(* CODESYS project TSR Libary.library
   Company: Eaton Automation
   Title: TSR Libary
   Description: Das ist eine Libary die die Wichtigsten Funktionen für den Touch-Simulations Roboter berteitstellt.
   Author: Samuel A. Marti
   Version: 1.3

Project tree, tasks and I/O mapping:
  libraries: Standard, 3.5.2.0 (System); CAA SerialCom, 3.5.3.0 (CAA Technical Workgroup)
  POUs/
    TSR Com/
      function block TSR_Com [ST]: A00_Start, A01_Get_Settings, A02_Open_Com, A03_Open_Wait, A04_Send_Com, A05_Send_Wait, A06_Receive_Com, A07_Receive_Wait, A08_String_Auswertung, A09_End, B0100_Error, A10_Start, A13_End, B1100_Error, A12_Close_Wait, A11_Close_Com, A0_Port_Senden, A1_Port_Schliessen
    FB Connect with TSR/
      function block Connect_with_TSR [ST]: B100_Error, A00_Start, A01_Progress, A02_Progress_Wait, A03_Auswerten, A04_End, A10_Start, A11_Progress, A12_Progress_Wait, A13_Auswerten, A14_End, A0_Connect_with_TSR, A1_Disconnect_with_TSR
    FN Set TSR startpoint/
      function FN_Set_TSR_startpoint [ST]
    FB Move TSR xy/
      function block FB_Move_TSR_xy [ST]: A0_Start, A1_Progress, A2_Progress_Wait, A3_Auswerten, A4_Wait_for_TSR, A5_Wait_for_TSR_Wait, A6_Wait_for_TSR_Auswerten, A7_End, B100_Error
    FB Go to TSR xy/
      function block FB_Go_to_TSR_xy [ST]: A0_Start, A1_Progress, A2_Progress_Wait, A3_Auswerten, A4_Wait_for_TSR, A5_Wait_for_TSR_Wait, A6_Wait_for_TSR_Auswerten, A7_End, B100_Error
    FB Get TSR position/
      function block FB_Get_TSR_position [ST]: A0_Start, A1_Progress, A2_Progress_Wait, A3_Auswerten, A4_End, B100_Error
    FB TSR Pen up down/
      function block TSR_Pen_up_down [ST]: A0_Start, A1_Progress, A2_Progress_Wait, A3_Auswerten, A4_End, B100_Error
    FB Click/
      function block FB_Click [ST]: A0_Start, A1_Progress, A2_Progress_Wait, A3_PenDown, A4_PenDown_Wait, A5_PenUp, A6_PenUp_Wait, A7_End, B100_Error
    FB Double Click/
      function block FB_Double_Click [ST]: A0_Start, A1_Progress, A2_Progress_Wait, A3_PenDown, A4_PenDown_Wait, A5_PenUp, A6_PenUp_Wait, A7_End, B100_Error
  global variables GLOBAL
*)

// GLOBAL
VAR_GLOBAL
iStartPosx				:INT;			//Die Globale Variable des Neuen nulpunkts für die anderen FB's
iStartPosy				:INT;			//""
GTr_Faktor				:REAL := 8.8;	//Der umrechnungs Faktor: Momentan ist er auf mm abgestummen.
FB_TSRCom: 				TSR_Com;		//Die Com Communication
END_VAR

// POUs/TSR Com/TSR_Com
FUNCTION_BLOCK TSR_Com
VAR_INPUT									//FB Eingänge	
	xExecute				:BOOL;				//Startbedingung für den FB.
	iCom					:INT;				//Die Nummer des Com Ports.
	stSendData				:STRING;			//Der String der Gesendet werden soll.
	xPort					:BOOL;				//Wenn = 0 Wird der Port geschlossen, Wenn = 1 Wird der Port geöffnet.
END_VAR

VAR_OUTPUT									//FB Ausgänge
	xBusy					:BOOL;				//Das Busy bit.
	xDone					:BOOL;				//Ist 1 wenn FB fertig ist.
	stReceivedData			:STRING;			//Der Empfangene Daten String.
	wState					:WORD;				//Der ENUM Wert für die ENUM Tabelle.
	xError					:BOOL;				//Ist 1 wenn es einen Error gab.
END_VAR

VAR											//Interne Var
	LTi_Zustand				:INT;				//Der Zustand.
	LTi_PosString			:INT;				//Die Position vom Carisch retain lengfield.
	LTocpa_ComParameter1	:ARRAY[1..20] OF COM.PARAMETER; //Initalisierung der Com Parameter.
	
	LTx_ComOpen				:BOOL;				//Gibt an ob ein Com Port schon offen ist.
	LTudi_Handle			:UDINT;				//Der Interne COM Handle.
	LTst_ReceivedData		:STRING;			//Received Data zwischenspeicher.

	LTfb_ComOpen			:Com.Open;			//FB Open.
	LTfb_WriteCom			:Com.Write;			//FB Write.
	LTfb_ReadCom			:Com.Read;			//FB Read.
	LTfb_Close				:Com.Close;			//FB Für den Com port zu schliessen.
	LTfb_Timer				:TON;				//Timer Init.
	
	LTudi_ComPort			:UDINT;				//Welcher Com Port ist gemeint.

END_VAR

VAR CONSTANT								//Konstanten, Einstellungen
	LCudi_StopBit			:UDINT := 0;		//Die Stopbits: 0 = 1stb, 1 = 1.5stb, 2 = 2stb.
	LCudi_Parity			:UDINT := 2;		//Parity: 0 = gerade, 1 = ungerade, 2 = keine.
	LCudi_Baudrate			:UDINT := 9600; 	//Möglich sind 2,5 m 115200 Bit/s, 5 m 57600 Bit/s, 10 m 38400 Bit/s, 15 m 19200 Bit/s, 30 m 9600 Bit/s
	LCudi_TimeOut			:UDINT := 0;		//Keine ahnung was das bewirkt.
	LCudi_BufferSize		:UDINT := 2048;		//Die Buffer grösse.
	LCudi_ByteSize			:UDINT := 8;		//Die Grösse vom daten Byte. kann nur von 4 bis 8 sein
	LCudi_Binary			:UDINT := 0;		//Binärmodus, keine EOF-Überprüfung/ keine ahnung wad das ist.
	LCudi_OutxCTSFlow		:UDINT := 0;		//CTS Handshake auf Ausgang/ keine ahnung wad das ist.
	LCudi_OutxDSRFlow		:UDINT := 0; 		//DSR Handshake auf Ausgang/ keine ahnung wad das ist.
	LCudi_DTRControl		:UDINT := 0;		//DTR Control. DTR Flusssteuerung/ keine ahnung wad das ist.
	LCudi_DSRSensitiv		:UDINT := 0; 		//DSR Empfindlichkeit/ keine ahnung wad das ist.
	LCudi_RTSControl		:UDINT := 0;		//Rts Flussteuerung/ keine ahnung wad das ist.
	LCudi_TXContinueOnXoff	:UDINT := 0;		//XOFF fortfahren Tx / keine ahnung wad das ist.
	LCudi_OUTX				:UDINT := 0;		//XON/XOFF Ausgabeflusssteuerung / keine ahnung wad das ist.
	LCudi_INX				:UDINT := 0;		//XON/XOFF Eingabeflusssteuerung / keine ahnung wad das ist.
	LCudi_XOnChar			:UDINT := 0;		//Tx AND Rx XON Zeichen / keine ahnung wad das ist.
	LCudi_XOffChar			:UDINT := 0;		//Tx AND Rx XOFF Zeichen.
	LCudi_XOnLim			:UDINT := 0;		//Übertrage XON Schwellenwert
	LCudi_XOffLim			:UDINT := 0;		//Übertrage XOFF Schwellenwert
	
	LCt_WaitTimeout			:TIME := T#4S;			//der Timout Timer.
	LCt_WaitCom				:TIME := T#600MS;		//Wait auf Received Data.
END_VAR

IF xPort = 1 THEN
	A0_Port_Senden();
END_IF

IF xPort = 0 THEN
	A1_Port_Schliessen();
END_IF

LTfb_Close();
LTfb_ComOpen();

ACTION A00_Start:
IF xExecute THEN			//Prüfe Startbedinung.
	xBusy := 1;				//Setze Busy.
	IF LTx_ComOpen THEN 	//Ist der Com Port offen ?
		LTi_Zustand := 4;	//Gehe direkt zum Schritt wo der String geschrieben wird.
	ELSE
		LTi_Zustand := 1;	//Gehe direkt zum Schritt wo der Com Port geöffnet wird.
	END_IF
END_IF
END_ACTION

ACTION A01_Get_Settings:
LTudi_ComPort := INT_TO_UDINT(iCom);

//Port
LTocpa_ComParameter1[1].udiParameterId := COM.CAA_Parameter_Constants.udiPort;		//ID von Com Port
LTocpa_ComParameter1[1].udiValue := LTudi_ComPort;									//Der COM Port1

//Stopbit
LTocpa_ComParameter1[2].udiParameterId := COM.CAA_Parameter_Constants.udiStopBits;	//ID von StopBit
LTocpa_ComParameter1[2].udiValue := LCudi_StopBit;									//Der COM Port. 0 = 1stb, 1 = 1.5stb, 2 = 2stb.

//Parität
LTocpa_ComParameter1[3].udiParameterId := COM.CAA_Parameter_Constants.udiParity;		//ID von Parity
LTocpa_ComParameter1[3].udiValue := LCudi_Parity;									//0 = gerade, 1 = ungerade, 2 = keine.

//Baudrate
LTocpa_ComParameter1[4].udiParameterId := COM.CAA_Parameter_Constants.udiBaudrate;	//ID von Baudrate
LTocpa_ComParameter1[4].udiValue := LCudi_Baudrate;									//Möglich sind 2,5 m 115200 Bit/s, 5 m 57600 Bit/s, 10 m 38400 Bit/s, 15 m 19200 Bit/s, 30 m 9600 Bit/s

//Timeout
LTocpa_ComParameter1[5].udiParameterId := COM.CAA_Parameter_Constants.udiTimeout;	//ID von Timeout
LTocpa_ComParameter1[5].udiValue := LCudi_TimeOut;									//Keine ahnung wad das ist.
(*
//BufferSize																		
LTocpa_ComParameter1[6].udiParameterId := COM.CAA_Parameter_Constants.udiBufferSize;	//ID von Buffersize
LTocpa_ComParameter1[6].udiValue := GLRudi_BufferSize;								//Die Grösse die der Buffer haben soll
*)
//ByteSize																	
LTocpa_ComParameter1[7].udiParameterId := COM.CAA_Parameter_Constants.udiByteSize;	//ID von ByteSize
LTocpa_ComParameter1[7].udiValue := LCudi_ByteSize;									//Die Grösse vom daten Byte. kann nur von 4 bis 8 sein

//Binary
LTocpa_ComParameter1[8].udiParameterId := COM.CAA_Parameter_Constants.udiBinary;	//ID von Binary
LTocpa_ComParameter1[8].udiValue := LCudi_Binary;									//Binärmodus, keine EOF-Überprüfung/ keine ahnung wad das ist.
(*
//OutxCtsFlow
LTocpa_ComParameter1[9].udiParameterId := COM.CAA_Parameter_Constants.udiOutxCtsFlow;	//ID von OutxCtsFlow
LTocpa_ComParameter1[9].udiValue := LCudi_OutxCTSFlow;									//CTS Handshake auf Ausgang/ keine ahnung wad das ist.

//OutxDSRFlow
LTocpa_ComParameter1[10].udiParameterId := COM.CAA_Parameter_Constants.udiOutxDsrFlow;	//ID von OutxDSRFlow
LTocpa_ComParameter1[10].udiValue := LCudi_OutxDSRFlow;									//DSR Handshake auf Ausgang/ keine ahnung wad das ist.

//DTRControl
LTocpa_ComParameter1[11].udiParameterId := COM.CAA_Parameter_Constants.udiDtrControl;	//ID von DtrControl
LTocpa_ComParameter1[11].udiValue := LCudi_OutxDSRFlow;									//DSR Handshake auf Ausgang/ keine ahnung wad das ist.

//DSR Sensitiv
LTocpa_ComParameter1[12].udiParameterId := COM.CAA_Parameter_Constants.udiDsrSensitivity;//ID von DSR Sensitiv
LTocpa_ComParameter1[12].udiValue := LCudi_DSRSensitiv;									//DSR Empfindlichkeit/ keine ahnung wad das ist.

//RTS Control
LTocpa_ComParameter1[13].udiParameterId := COM.CAA_Parameter_Constants.udiRtsControl;	//ID von RTS Control
LTocpa_ComParameter1[13].udiValue := LCudi_RTSControl;									//Rts Flusssteuerung/ keine ahnung wad das ist.

//TXContinueOnXoff	
LTocpa_ComParameter1[14].udiParameterId := COM.CAA_Parameter_Constants.udiTXContinueOnXoff;	//ID von  XOFF fortfahren Tx	
LTocpa_ComParameter1[14].udiValue := LCudi_TXContinueOnXoff;									//XOFF fortfahren Tx / keine ahnung wad das ist.

//OUT X
LTocpa_ComParameter1[15].udiParameterId := COM.CAA_Parameter_Constants.udiOutX;	//ID von OUT X	
LTocpa_ComParameter1[15].udiValue := LCudi_OUTX;									//XON/XOFF Ausgabeflusssteuerung/ keine ahnung wad das ist.

//IN X
LTocpa_ComParameter1[16].udiParameterId := COM.CAA_Parameter_Constants.udiInX;	//ID von IN X	
LTocpa_ComParameter1[16].udiValue := LCudi_INX;									//Eingabeflusssteuerung/ keine ahnung wad das ist.

//XOnChar
LTocpa_ComParameter1[17].udiParameterId := COM.CAA_Parameter_Constants.udiXonChar;	//ID von x on char	
LTocpa_ComParameter1[17].udiValue := LCudi_XOnChar;									//Tx AND Rx XON Zeichen/ keine ahnung wad das ist.

//XOffChar
LTocpa_ComParameter1[18].udiParameterId := COM.CAA_Parameter_Constants.udiXoffChar;	//ID von x off char
LTocpa_ComParameter1[18].udiValue := LCudi_XOffChar;									//Tx AND Rx XOFF Zeichen/ keine ahnung wad das ist.

//XonLim
LTocpa_ComParameter1[19].udiParameterId := COM.CAA_Parameter_Constants.udiXonLim;	//ID von X on Lim
LTocpa_ComParameter1[19].udiValue := LCudi_XOnLim;									//Übertrage XON Schwellenwert/ keine ahnung wad das ist.

//XoffLim
LTocpa_ComParameter1[20].udiParameterId := COM.CAA_Parameter_Constants.udiXonLim;	//ID von X off Lim
LTocpa_ComParameter1[20].udiValue := LCudi_XOnLim;									//Übertrage XOFF Schwellenwert/ keine ahnung wad das ist.
*)
LTi_Zustand := 2;
END_ACTION

ACTION A02_Open_Com:
//Com Port öffnen
LTfb_ComOpen.usiListLength := INT_TO_USINT(SIZEOF(LTocpa_ComParameter1));	//Die länge der Parameter Liste
LTfb_ComOpen.pParameterList := ADR(LTocpa_ComParameter1);		//Die Adresse der Parameter Liste
LTfb_ComOpen.xExecute := 1;									//Start Flag setzten.
LTi_Zustand := 3;
LTfb_Timer(IN := 1, PT:= LCt_WaitTimeout);								//Rufe Timer auf
END_ACTION

ACTION A03_Open_Wait:
IF LTfb_ComOpen.xDone THEN											//Wenn der Port offen
	LTfb_Timer.IN := 0;					//Timer Zurücksetzten.
	LTi_Zustand := 4;					//Gehe in den Sende Schritt
	LTudi_Handle := LTfb_ComOpen.hCom;	//Speichere den Handle
	LTx_ComOpen	:= 1;					//Der Offene Com Port setzten.
ELSE
	IF LTfb_ComOpen.xError THEN				//Wenn es einen Error bei Com Port öffnen gab.
		LTfb_Timer.IN := 0;					//Timer Zurücksetzten.
		LTi_Zustand := 100;					//In den Error Zustand gehen.
		wState := 1;						//Den ENUM Wert Error angeben.
	ELSE
		IF LTfb_Timer.Q THEN						//Wenn der Timer Abgelaufen ist.
			LTi_Zustand := 100;					//In den Error Zustand gehen.
			wState := 4;						//Den ENUM Wert Error angeben.
			LTfb_Timer.IN := 0;
		END_IF
	END_IF
END_IF

LTfb_Timer();								//Rufe Timer auf
LTfb_ComOpen();							//Rufe den FB auf.
END_ACTION

ACTION A04_Send_Com:
LTfb_WriteCom(
	hCom			:= LTudi_Handle, 						//Ubergebe Handle.
	pBuffer 		:= ADR(stSendData),
	szSize 			:= INT_TO_UDINT(SIZEOF(stSendData)),
	xExecute		:= 1									//Starte Sende Vorgang.
);

LTi_Zustand := 5;
LTfb_Timer(IN := 1, PT:= LCt_WaitTimeout);				//Rufe Timer auf
END_ACTION

ACTION A05_Send_Wait:
IF LTfb_WriteCom.xDone THEN				//Wenn der String gesendet wurde.
	LTfb_Timer.IN := 0;					//Timer Zurücksetzten.
	LTi_Zustand := 6;					//Gehe in den Sende Schritt
ELSE
	IF LTfb_WriteCom.xError THEN				//Wenn es einen Error bei String senden gab.
		LTfb_Timer.IN := 0;					//Timer Zurücksetzten.
		LTi_Zustand := 100;					//In den Error Zustand gehen.
		wState := 2;						//Den ENUM Wert Error angeben.
	ELSE
		IF LTfb_Timer.Q THEN						//Wenn der Timer Abgelaufen ist.
			LTi_Zustand := 100;					//In den Error Zustand gehen.
			wState := 5;						//Den ENUM Wert Error angeben.
			LTfb_Timer.IN := 0;
		END_IF
	END_IF
END_IF

LTfb_Timer();								//Rufe Timer auf
LTfb_WriteCom();							//Rufe den FB auf.
END_ACTION

ACTION A06_Receive_Com:
LTfb_Timer(IN := 1, PT:= LCt_WaitCom);			//Rufe Timer auf
IF LTfb_TIMER.Q THEN							//Wenn der Timer fertig ist
	LTfb_Timer.IN := 0;						//Timer zurücksetzten
	LTfb_Timer();								//FB Timer zurückstzen.
	
	LTfb_ReadCom								//Rufe ReadCom auf.
	(
		xExecute	:= 1,					//Starte Lese STRING
		hCom		:= LTudi_Handle,		//übergib den Handle.
		pBuffer := ADR(LTst_ReceivedData),
		szBuffer := SIZEOF(LTst_ReceivedData),
	);
LTi_Zustand := 7;

END_IF
END_ACTION

ACTION A07_Receive_Wait:
IF LTfb_ReadCom.xDone THEN				//Wenn der String gesendet wurde.
	LTfb_Timer.IN := 0;					//Timer Zurücksetzten.
	LTi_Zustand := 8;					//Gehe in den Sende Schritt
ELSE
	IF LTfb_ReadCom.xError THEN				//Wenn es einen Error bei String senden gab.
		LTfb_Timer.IN := 0;					//Timer Zurücksetzten.
		LTi_Zustand := 100;					//In den Error Zustand gehen.
		wState := 3;						//Den ENUM Wert Error angeben.
	ELSE
		IF LTfb_Timer.Q THEN						//Wenn der Timer Abgelaufen ist.
			LTi_Zustand := 100;					//In den Error Zustand gehen.
			wState := 6;						//Den ENUM Wert Error angeben.
			LTfb_Timer.IN := 0;
		END_IF
	END_IF
LTfb_Timer(IN := 1, PT:= LCt_WaitTimeout);			//Schalte Timer ein.
END_IF

LTfb_Timer();								//Rufe Timer auf
LTfb_ReadCom();							//Rufe den FB auf.
END_ACTION

ACTION A08_String_Auswertung:
LTi_PosString := FIND(STR2:='$R$N' , STR1:=LTst_ReceivedData);		//Das caretsch Retain lengfield 
LTst_ReceivedData[LTi_PosString - 1] := 0;							//DAs caretain legas löschen mit allem was dahinter ist.
stReceivedData := LTst_ReceivedData;								//Ausgeben
LTi_Zustand := 9;													//Zum Zustand 9 gehen.
END_ACTION

ACTION A09_End:
xBusy := 0;							//Alles zurücksetzten
xDone := 1;
IF xExecute = 0 THEN				//Warten bis der User Zurückgesetzt hat.
	xDone := 0;
	LTi_Zustand := 0;
	stReceivedData := '';
	LTfb_WriteCom.xExecute := 0;
	LTfb_ReadCom.xExecute := 0;
	LTst_ReceivedData := '';
	LTfb_ComOpen.xExecute := 0;
	LTfb_WriteCom();
	LTfb_ReadCom();
	LTfb_ComOpen();
END_IF
END_ACTION

ACTION B0100_Error:
xBusy := 0;							//Alles zurücksetzten
xError := 1;
IF xExecute = 0 THEN				//Wartem bis der User das xExecute zurückgesetzt hat.
	xError := 0;
	LTi_Zustand := 0;
	wState := 0;
	stReceivedData := '';
	LTst_ReceivedData := '';
	LTfb_WriteCom.xExecute := 0;
	LTfb_ReadCom.xExecute := 0;
	LTfb_ComOpen.xExecute := 0;
	LTfb_WriteCom();
	LTfb_ReadCom();
	LTfb_ComOpen();
END_IF
END_ACTION

ACTION A10_Start:
IF xExecute THEN			//Prüfe Startbedinung.
	xBusy := 1;				//Setze Busy.
	IF LTx_ComOpen THEN 	//Ist der Com Port offen ?
		LTi_Zustand := 1;	//Gehe direkt zum Schritt wo der String geschrieben wird.
	ELSE
		LTi_Zustand := 100; //Gehe in den Error Mod
		wState := 13;		//Bedeutung: Der com port ist nicht offen daher kann nichts geschlossen werden. 		
	END_IF
END_IF
END_ACTION

ACTION A13_End:
xBusy := 0;							//Alles zurücksetzten
xDone := 1;
IF xExecute = 0 THEN				//Warten bis der User Zurückgesetzt hat.
	xDone := 0;
	LTi_Zustand := 0;
	stReceivedData := '';
	LTst_ReceivedData := '';
	LTfb_Close.xExecute := 0;
	LTfb_Close();
END_IF
END_ACTION

ACTION B1100_Error:
xBusy := 0;							//Alles zurücksetzten
xError := 1;
IF xExecute = 0 THEN				//Wartem bis der User das xExecute zurückgesetzt hat.
	xError := 0;
	LTi_Zustand := 0;
	wState := 0;
	stReceivedData := '';
	LTst_ReceivedData := '';
	LTfb_Close.xExecute := 0;
	LTfb_Close();
END_IF
END_ACTION

ACTION A12_Close_Wait:
IF LTfb_Close.xDone THEN											//Wenn der Port offen
	LTfb_Timer.IN := 0;					//Timer Zurücksetzten.
	LTi_Zustand := 3;					//Gehe in den Finish schritt.
	LTx_ComOpen := 0;					//Denn Das Com Port flag zurücksetzten.
ELSE
	IF LTfb_Close.xError THEN				//Wenn es einen Error bei Com Port öffnen gab.
		LTfb_Timer.IN := 0;					//Timer Zurücksetzten.
		LTi_Zustand := 100;					//In den Error Zustand gehen.
		wState := 23;						//Den ENUM Wert Error angeben.
	ELSE
		IF LTfb_Timer.Q THEN						//Wenn der Timer Abgelaufen ist.
			LTi_Zustand := 100;					//In den Error Zustand gehen.
			wState := 24;						//Den ENUM Wert Error angeben.
			LTfb_Timer.IN := 0;
		END_IF
	END_IF
END_IF

LTfb_Timer();								//Rufe Timer auf
LTfb_ComOpen();							//Rufe den FB auf.
END_ACTION

ACTION A11_Close_Com:
LTfb_Close
(
	xExecute := 1 , 			//Setzt den Zustand vom Execute auf 1.
	hCom := LTudi_Handle, 		//übergebe den Handle des geöffneten Com Ports.
);
LTi_Zustand := 2;
END_ACTION

ACTION A0_Port_Senden:
CASE LTi_Zustand OF
	0:
		A00_Start();					//Prüfe die Startbedingungen und Prüfe auf einen offenen Com Port
	1:
		A01_Get_Settings();			//Holt die Einstellungen für zu öffnenden Com Port.
	2:
		A02_Open_Com();				//Öffnet den Com Port.
	3:
		A03_Open_Wait();				//Wartet bis der Com Port offen ist.
	4:
		A04_Send_Com();				//Den String Senden.
	5:
		A05_Send_Wait();				//Warte bis der String gesendet wurde.
	6:
		A06_Receive_Com();			//Empfange den String.
	7:
		A07_Receive_Wait();			//Warte auf FB String lesen.
	8:
		A08_String_Auswertung();		//Werte den FB String aus.
	9:
		A09_End();					//Beende den FB vorgang und warte auf das zurücksetzten.
	100:
		B0100_Error();				//Nur wenn ein Error gab.
END_CASE

LTfb_ComOpen();
END_ACTION

ACTION A1_Port_Schliessen:
CASE LTi_Zustand OF
	0:
		A10_Start();					//Prüfe die Startbedingungen und Prüfe auf einen offenen Com Port.
	1:
		A11_Close_Com();				//schliesst den Com Port.
	2:
		A12_Close_Wait();				//Warten bis der Com Port geschlossen.
	3:
		A13_End();						//Beendet den schliess vorgang.
	100:
		B1100_Error();					//Der Error Modus.
END_CASE

LTfb_Close();
END_ACTION

END_FUNCTION_BLOCK

// POUs/FB Connect with TSR/Connect_with_TSR
FUNCTION_BLOCK Connect_with_TSR
VAR_INPUT								//FB Eingänge
	xExecute				:BOOL;			//Startbedingung für den FB.
	iCom					:INT;			//Die Nummer des Com Ports.
	xPort					:BOOL;			//Bei 0 = den Port schliessen, bei 1 = Prot öffnen.
END_VAR

VAR_OUTPUT								//FB Ausgänge	
	xBusy					:BOOL;			//Das Busy bit.
	xDone					:BOOL;			//Ist 1 wenn FB fertig ist.
	wState					:WORD;			//Der ENUM Wert für die ENUM Tabelle.
	xError					:BOOL;			//Ist 1 wenn es einen Error gab.
END_VAR

VAR										//Interne Vars
	LTi_Zustand				:INT;			//Der Zustand.
	GLfb_Timer				:TON;			//Timer Init
END_VAR

VAR CONSTANT							//Konstanten, Einstellungen
	LCt_WaitTimeout			:TIME := T#4S;	//der Timout Timer. Nach welcher Zeit soll es einen Timeout geben.
END_VAR

//Entscheiden ob der COM Port geöffnent werden soll oder geschlossen werden soll
IF xPort = 0 THEN
	A1_Disconnect_with_TSR();	//Verbindung Abbrechen
END_IF

IF xPort = 1 THEN
	A0_Connect_with_TSR();		//Verbindung herstellen
END_IF
FB_TSRCom();

ACTION B100_Error:
xBusy := 0;							//Alles zurücksetzten
xError := 1;
IF xExecute = 0 THEN				//Wartem bis der User das xExecute zurückgesetzt hat.
	xError := 0;
	LTi_Zustand := 0;
	wState := 0;
	FB_TSRCom.xEXecute := 0;
END_IF
END_ACTION

ACTION A00_Start:
IF xExecute THEN			//Prüfe Startbedinung.
	xBusy := 1;				//Setze Busy.
	LTi_Zustand := 1;	//Gehe direkt zum Schritt wo der Com Port geöffnet wird.
END_IF
END_ACTION

ACTION A01_Progress:
FB_TSRCom(						//TSR Com Aufrufen und Daten übergeben.
	xEXecute	:=	1 , 
	xPort		:=	xPort,
	iCom		:= 	iCom, 
	stSendData	:= 	'?',  );
LTi_Zustand := 2;				//In den nächsten Zustand Wechseln.
END_ACTION

ACTION A02_Progress_Wait:
IF FB_TSRCom.xDone THEN											//Wenn der Port offen
	GLfb_Timer.IN := 0;					//Timer Zurücksetzten.
	LTi_Zustand := 3;					//Gehe in den Sende Schritt
ELSE
	IF FB_TSRCom.xError THEN				//Wenn es einen Error bei Com Port öffnen gab.
		GLfb_Timer.IN := 0;					//Timer Zurücksetzten.
		LTi_Zustand := 100;					//In den Error Zustand gehen.
		wState := FB_TSRCom.wState;			//Den ENUM Wert Error angeben.
	ELSE
		IF GLfb_Timer.Q THEN						//Wenn der Timer Abgelaufen ist.
			LTi_Zustand := 100;					//In den Error Zustand gehen.
			wState := 16;						//Timeout beim Connect
			GLfb_Timer.IN := 0;
		END_IF
	END_IF
GLfb_Timer(IN := 1, PT:= LCt_WaitTimeout);
END_IF

GLfb_Timer();								//Rufe Timer auf
END_ACTION

ACTION A03_Auswerten:
IF FB_TSRCom.stReceivedData = '!' THEN		//Wenn der TSR reagiert.
	LTi_Zustand := 4;						//Gehe zum letzten Zustand.
ELSE											
	LTi_Zustand := 100;	
	wState := 8;								
END_IF
END_ACTION

ACTION A04_End:
xBusy := 0;							//Alles zurücksetzten
xDone := 1;
IF xExecute = 0 THEN				//Warten bis der User Zurückgesetzt hat.
	xDone := 0;
	LTi_Zustand := 0;
	FB_TSRCom.xEXecute := 0;
END_IF
END_ACTION

ACTION A10_Start:
IF xExecute THEN			//Prüfe Startbedinung.
	xBusy := 1;				//Setze Busy.
	LTi_Zustand := 1;	//Gehe direkt zum Schritt wo der Com Port geöffnet wird.
END_IF
END_ACTION

ACTION A11_Progress:
FB_TSRCom(						//TSR Com Aufrufen und Daten übergeben.
	xEXecute	:=	1 , 
	iCom		:= 	iCom, 
	xPort		:=	xPort, );
LTi_Zustand := 2;				//In den nächsten Zustand Wechseln.
END_ACTION

ACTION A12_Progress_Wait:
IF FB_TSRCom.xDone THEN											//Wenn der Port offen
	GLfb_Timer.IN := 0;					//Timer Zurücksetzten.
	LTi_Zustand := 3;					//Gehe in den Sende Schritt
ELSE
	IF FB_TSRCom.xError THEN				//Wenn es einen Error bei Com Port öffnen gab.
		GLfb_Timer.IN := 0;					//Timer Zurücksetzten.
		LTi_Zustand := 100;					//In den Error Zustand gehen.
		wState := FB_TSRCom.wState;			//Den ENUM Wert Error angeben.
	ELSE
		IF GLfb_Timer.Q THEN					//Wenn der Timer Abgelaufen ist.
			LTi_Zustand := 100;					//In den Error Zustand gehen.
			wState := 16;						//Timeout_beim_Connect_weahrend_dem_TSR_COM
			GLfb_Timer.IN := 0;
		END_IF
	END_IF
GLfb_Timer(IN := 1, PT:= LCt_WaitTimeout);
END_IF

GLfb_Timer();								//Rufe Timer auf
END_ACTION

ACTION A13_Auswerten:
IF FB_TSRCom.stReceivedData = '' THEN		//Wenn der TSR reagiert.
	LTi_Zustand := 4;						//Gehe zum letzten Zustand.
ELSE											
	LTi_Zustand := 100;	
	wState := 8;								
END_IF
END_ACTION

ACTION A14_End:
xBusy := 0;							//Alles zurücksetzten
xDone := 1;
IF xExecute = 0 THEN				//Warten bis der User Zurückgesetzt hat.
	xDone := 0;
	LTi_Zustand := 0;
	FB_TSRCom.xEXecute := 0;
END_IF
END_ACTION

ACTION A0_Connect_with_TSR:
CASE LTi_Zustand OF
	0:
		A00_Start();					//Prüfe die Startbedingungen 
	1:
		A01_Progress();				//Starte den Prozess.
	2:
		A02_Progress_Wait();			//Warte auf den FB TSR Com
	3:
		A03_Auswerten();				//Werte das Egebniss aus.
	4:
		A04_End();					//Warte auf Execute
	100:
		B100_Error();				//Nur wenn ein Error gab.
END_CASE
END_ACTION

ACTION A1_Disconnect_with_TSR:
CASE LTi_Zustand OF
	0:
		A10_Start();					//Prüfe die Startbedingungen 
	1:
		A11_Progress();				//Starte den Prozess.
	2:
		A12_Progress_Wait();			//Warte auf den FB TSR Com
	3:
		A13_Auswerten();				//Werte das Egebniss aus.
	4:
		A14_End();					//Warte auf Execute
	100:
		B100_Error();				//Nur wenn ein Error gab.
END_CASE
END_ACTION

END_FUNCTION_BLOCK

// POUs/FN Set TSR startpoint/FN_Set_TSR_startpoint
FUNCTION FN_Set_TSR_startpoint : BOOL
VAR_INPUT							//FB EINGANGS VAR
	iStartpointx			:INT;		//Der Virtuelle x Nullpunkt.
	iStartpointy			:INT;		//Der Virtuelle y Nullpunkt.
END_VAR

iStartPosx := REAL_TO_INT(INT_TO_REAL(iStartpointx) * GTr_Faktor);		//Speicher eingang in Global Var
iStartPosy := REAL_TO_INT(INT_TO_REAL(iStartpointy) * GTr_Faktor);		//Speicher eingang in Global Var
FN_Set_TSR_startpoint := 1;												// Der Rückgabe wert der Funktion

END_FUNCTION

// POUs/FB Move TSR xy/FB_Move_TSR_xy
FUNCTION_BLOCK FB_Move_TSR_xy
VAR_INPUT									//Eingänge Var						
	xExecute				:BOOL;				//Startbedingung für den FB.
	iMovx					:INT;				//Die relative x bewegung des TSR in richtung x
	iMovy					:INT;				//Die relative y bewegung des TSR in richtung y
END_VAR

VAR_OUTPUT									//Ausgänge Var
	xBusy					:BOOL;				//Das Busy bit.
	xDone					:BOOL;				//Ist 1 wenn FB fertig ist.
	wState					:WORD;				//Der ENUM Wert für die ENUM Tabelle.
	xError					:BOOL;				//Ist 1 wenn es einen Error gab.
END_VAR

VAR											//Interne Var
	LTi_Zustand				:INT;				//Der Zustand.
	LTst_Zwischenspeicher	:STRING;			//Ein Zwischenspeicher für den Progress.
	LTi_Len					:INT;				//Gibt die String länge an für den Progress.
	LTi_x					:INT;				//Die x Schritte die der TSR machen soll.
	LTi_y					:INT;				//Die y Schritte die der TSR machen soll.
											//TIMER
	FN_Timer				:TON;				//Timer Init.
END_VAR

VAR CONSTANT								//Konstanten, Einstellungen
	LCt_WaitTimeout			:TIME := T#2S;		//der Timout Timer.
	LCt_WaitCom				:TIME := T#250MS;	//Wait auf Received Data.
END_VAR

CASE LTi_Zustand OF
	0:
		A0_Start();						//Prüfe Startbedingunen
	1:
		A1_Progress();					//Starte den Prozess. und sende den Befehl an das TSR.
	2:
		A2_Progress_Wait();				//Warte auf den FB Com.
	3:
		A3_Auswerten();					//Beende den FB und warte auf den User.
	4:
		A4_Wait_for_TSR();				//Init warten bis der TSR bei der Position angekommen ist
	5:
		A5_Wait_for_TSR_Wait();			//Warte auf FB Com.
	6:
		A6_Wait_for_TSR_Auswerten();	//Werte aus.
	7:
		A7_End();						//Das ende der Funktion.
	100:
		B100_Error();					//Die Error Aktion.
END_CASE

FB_TSRCom();							//Aufrufen.

ACTION A0_Start:
IF xExecute THEN			//Prüfe Startbedinung.
	xBusy := 1;				//Setze Busy.
	LTi_Zustand := 1;		//nächster Schritt
END_IF
END_ACTION

ACTION A1_Progress:
//Hier wird der Befehl für den TSR zusammengesetzt.
LTst_Zwischenspeicher := 'mov ';	//Speicher

//Die Fakto miteinbeziehen so das die mm umgerechnet werden, in Schritte.
LTi_x := REAL_TO_INT(INT_TO_REAL(iMovx) * GTr_Faktor);
//Schreibe Die X koordinate hinein.
LTst_Zwischenspeicher := INSERT(LTst_Zwischenspeicher,INT_TO_STRING(LTi_x),4); 

//Finde die länge des String heraus
LTi_Len := LEN(STR := LTst_Zwischenspeicher);

//Schreibe am Schluss ein :
LTst_Zwischenspeicher := INSERT(LTst_Zwischenspeicher,':',LTi_Len);

//Die Fakto miteinbeziehen so das die mm umgerechnet werden, in Schritte.
LTi_y := REAL_TO_INT(INT_TO_REAL(iMovy) * GTr_Faktor);
//Nun schreibe hinter dem : die y Koordiante.
LTst_Zwischenspeicher := INSERT(LTst_Zwischenspeicher,INT_TO_STRING(LTi_y),(LTi_Len + 1));

//TSR Com Aufrufen und Daten übergeben.
FB_TSRCom(						
	iCom		:= 1,
	xEXecute	:=	1 , 
	stSendData	:= 	LTst_Zwischenspeicher,  );

//Auf zum nächsten schritt.
LTi_Zustand := 2;
END_ACTION

ACTION A2_Progress_Wait:
IF FB_TSRCom.xDone THEN											//Wenn der Port offen
	FN_Timer.IN := 0;						//Timer Zurücksetzten.
	LTi_Zustand := 3;						//Gehe in den Sende Schritt
ELSE
	IF FB_TSRCom.xError THEN				//Wenn es einen Error bei Com Port öffnen gab.
		FN_Timer.IN := 0;					//Timer Zurücksetzten.
		LTi_Zustand := 100;					//In den Error Zustand gehen.
		wState := FB_TSRCom.wState;			//Den ENUM Wert Error angeben.
	ELSE
		IF FN_Timer.Q THEN					//Wenn der Timer Abgelaufen ist.
			LTi_Zustand := 100;				//In den Error Zustand gehen.
			wState := 21;					//Den ENUM Wert Error angeben.
			FN_Timer.IN := 0;
		END_IF
	END_IF
FN_Timer(IN := 1, PT:= LCt_WaitTimeout);	//Setzte den Timer.
END_IF
FN_Timer();									//Timer Aufrufen.
END_ACTION

ACTION A3_Auswerten:
IF FB_TSRCom.stReceivedData = 'moving' THEN //Wenn der TSR reagiert.
	LTi_Zustand := 4;						//Gehe zum letzten Zustand.
	FB_TSRCom.xEXecute := 0;				//Setzte Com Communication zurück.
ELSE
	IF FB_TSRCom.stReceivedData = 'out of range' THEN
		wState := 9;						//out of range state
		LTi_zustand := 100;
	ELSE
		LTi_Zustand := 100;
		wState := 8;							//Gehe zum letzten Zustand.
	END_IF
END_IF
END_ACTION

ACTION A4_Wait_for_TSR:
//TSR Com Aufrufen und Daten übergeben.
FB_TSRCom(						
	iCom		:= 1,
	xEXecute	:=	1 , 
	stSendData	:= 'state',  );				//frage den Status ab.

//Auf zum nächsten schritt.
LTi_Zustand := 5;
END_ACTION

ACTION A5_Wait_for_TSR_Wait:
IF FB_TSRCom.xDone THEN											//Wenn der Port offen
	FN_Timer.IN := 0;						//Timer Zurücksetzten.
	LTi_Zustand := 6;						//Gehe in den Sende Schritt
ELSE
	IF FB_TSRCom.xError THEN				//Wenn es einen Error bei Com Port öffnen gab.
		FN_Timer.IN := 0;					//Timer Zurücksetzten.
		LTi_Zustand := 100;					//In den Error Zustand gehen.
		wState := FB_TSRCom.wState;			//Den ENUM Wert Error angeben.
	ELSE
		IF FN_Timer.Q THEN					//Wenn der Timer Abgelaufen ist.
			LTi_Zustand := 100;				//In den Error Zustand gehen.
			wState := 21;					//Den ENUM Wert Error angeben.
			FN_Timer.IN := 0;
		END_IF
	END_IF
FN_Timer(IN := 1, PT:= LCt_WaitTimeout);	//Setzte den Timer.
END_IF
FN_Timer();									//Timer Aufrufen.
END_ACTION

ACTION A6_Wait_for_TSR_Auswerten:
IF FB_TSRCom.stReceivedData = 'ready' THEN 		//Wenn der TSR reagiert.
	LTi_Zustand := 7;							//Gehe zum letzten Zustand.
	FB_TSRCom.xEXecute := 0;					//Setzte Com Communication zurück.
ELSE
	IF FB_TSRCom.stReceivedData = 'busy' THEN	//Wenn der TSR noch busy ist frage nochmal.
		FB_TSRCom.xEXecute := 0;				
		LTi_zustand := 4;
	ELSE
		IF FB_TSRCom.stReceivedData = '' THEN
			FB_TSRCom.xEXecute := 0;				
			LTi_zustand := 4;
		ELSE
			LTi_Zustand := 100;
			wState := 8;							//Gehe zum letzten Zustand.
		END_IF 
	END_IF
END_IF
END_ACTION

ACTION A7_End:
xBusy := 0;							//Alles zurücksetzten
xDone := 1;
IF xExecute = 0 THEN				//Warten bis der User Zurückgesetzt hat.
	xDone := 0;
	LTi_Zustand := 0;
	FB_TSRCom.xEXecute := 0;
END_IF
END_ACTION

ACTION B100_Error:
xBusy := 0;							//Alles zurücksetzten
xError := 1;
IF xExecute = 0 THEN				//Wartem bis der User das xExecute zurückgesetzt hat.
	xError := 0;
	LTi_Zustand := 0;
	wState := 0;					
	FB_TSRCom.xEXecute := 0;		//FB Com zurücksetzetn
END_IF
END_ACTION

END_FUNCTION_BLOCK

// POUs/FB Go to TSR xy/FB_Go_to_TSR_xy
FUNCTION_BLOCK FB_Go_to_TSR_xy
VAR_INPUT								//FB Eingänge
	xExecute				:BOOL;			//Startbedingung für den FB.
	iGotox					:INT;			//Die relative x bewegung des TSR in richtung x
	iGotoy					:INT;			//Die relative y bewegung des TSR in richtung y
END_VAR

VAR_OUTPUT								//FB Ausgänge
	xBusy					:BOOL;			//Das Busy bit.
	xDone					:BOOL;			//Ist 1 wenn FB fertig ist.
	wState					:WORD;			//Der ENUM Wert für die ENUM Tabelle.
	xError					:BOOL;			//Ist 1 wenn es einen Error gab.
END_VAR

VAR										//Interne Var
	LTi_Zustand				:INT;			//Der Zustand.
	LTst_Zwischenspeicher	:STRING;		//Ein Zwischenspeicher für den Progress.
	LTi_Len					:INT;			//Gibt die String länge an für den Progress.
	LTi_x					:INT;			//Die x Schritte die der TSR machen soll.
	LTi_y					:INT;			//Die y Schritte die der TSR machen soll.
										//TIMER
	LTfn_Timer				:TON;			//Timer Init.
END_VAR

VAR CONSTANT							//Konstanten, Einstellungen
	LCt_WaitTimeout			:TIME := T#2S;	//der Timout Timer.
	LCt_WaitCom				:TIME := T#250MS;//Wait auf Received Data.
END_VAR

CASE LTi_Zustand OF
	0:
		A0_Start();						//Prüfe Startbedingunen
	1:
		A1_Progress();					//Starte den Prozess. und sende den Befehl an das TSR.
	2:
		A2_Progress_Wait();				//Warte auf den FB Com.
	3:
		A3_Auswerten();					//Beende den FB und warte auf den User.
	4:
		A4_Wait_for_TSR();				//Init warten bis der TSR bei der Position angekommen ist
	5:
		A5_Wait_for_TSR_Wait();			//Warte auf FB Com.
	6:
		A6_Wait_for_TSR_Auswerten();	//Werte aus.
	7:
		A7_End();						//Das ende der Funktion.
	100:
		B100_Error();					//Die Error Aktion.
END_CASE

FB_TSRCom();							//Der COM muss hier nochmals aufgerufen werden weil er ansonten nicht hinterkommt.

ACTION A0_Start:
IF xExecute THEN			//Prüfe Startbedinung.
	xBusy := 1;				//Setze Busy.
	LTi_Zustand := 1;		//nächster Schritt
END_IF
END_ACTION

ACTION A1_Progress:
//Hier wird der Befehl für den TSR zusammengesetzt.
LTst_Zwischenspeicher := 'movto ';	//Speicher

//Die Fakto miteinbeziehen so das die mm umgerechnet werden, in Schritte.
LTi_x := iStartPosx + (REAL_TO_INT(INT_TO_REAL(iGotox) * GTr_Faktor));
//Schreibe Die X koordinate hinein.
LTst_Zwischenspeicher := INSERT(LTst_Zwischenspeicher,INT_TO_STRING(LTi_x),6); 

//Finde die länge des String heraus
LTi_Len := LEN(STR := LTst_Zwischenspeicher);

//Schreibe am Schluss ein :
LTst_Zwischenspeicher := INSERT(LTst_Zwischenspeicher,':',LTi_Len);

//Die Fakto miteinbeziehen so das die mm umgerechnet werden, in Schritte.
LTi_y := iStartPosy + (REAL_TO_INT(INT_TO_REAL(iGotoy) * GTr_Faktor));
//Nun schreibe hinter dem : die y Koordiante.
LTst_Zwischenspeicher := INSERT(LTst_Zwischenspeicher,INT_TO_STRING(LTi_y),(LTi_Len + 1));

//TSR Com Aufrufen und Daten übergeben.
FB_TSRCom
(						
	iCom		:= 1,
	xEXecute	:= 1 , 
	stSendData	:=  LTst_Zwischenspeicher,  
);

//Auf zum nächsten schritt.
LTi_Zustand := 2;
END_ACTION

ACTION A2_Progress_Wait:
IF FB_TSRCom.xDone THEN											//Wenn der Port offen
	LTfn_Timer.IN := 0;						//Timer Zurücksetzten.
	LTi_Zustand := 3;						//Gehe in den Sende Schritt
ELSE
	IF FB_TSRCom.xError THEN				//Wenn es einen Error bei Com Port öffnen gab.
		LTfn_Timer.IN := 0;					//Timer Zurücksetzten.
		LTi_Zustand := 100;					//In den Error Zustand gehen.
		wState := FB_TSRCom.wState;			//Den ENUM Wert Error angeben.
	ELSE
		IF LTfn_Timer.Q THEN				//Wenn der Timer Abgelaufen ist.
			LTi_Zustand := 100;				//In den Error Zustand gehen.
			wState := 20;					//Den ENUM Wert Error angeben.
			LTfn_Timer.IN := 0;
		END_IF
	END_IF
LTfn_Timer(IN := 1, PT:= LCt_WaitTimeout);	//Setzte den Timer.
END_IF
LTfn_Timer();								//Timer Aufrufen.
END_ACTION

ACTION A3_Auswerten:
IF FB_TSRCom.stReceivedData = 'moving' THEN //Wenn der TSR reagiert.
	LTi_Zustand := 4;						//Gehe zum letzten Zustand.
	FB_TSRCom.xEXecute := 0;				//Setzte Com Communication zurück.
ELSE
	IF FB_TSRCom.stReceivedData = 'out of range' THEN
		wState := 9;						//out of range state
		LTi_zustand := 100;
	ELSE
		LTi_Zustand := 100;
		wState := 8;							//Gehe zum letzten Zustand.
	END_IF
END_IF
END_ACTION

ACTION A4_Wait_for_TSR:
//TSR Com Aufrufen und Daten übergeben.
FB_TSRCom(						
	iCom		:= 1,
	xEXecute	:=	1 , 
	stSendData	:= 'state',  );				//frage den Status ab.

//Auf zum nächsten schritt.
LTi_Zustand := 5;
END_ACTION

ACTION A5_Wait_for_TSR_Wait:
IF FB_TSRCom.xDone THEN											//Wenn der Port offen
	LTfn_Timer.IN := 0;						//Timer Zurücksetzten.
	LTi_Zustand := 6;						//Gehe in den Sende Schritt
ELSE
	IF FB_TSRCom.xError THEN				//Wenn es einen Error bei Com Port öffnen gab.
		LTfn_Timer.IN := 0;					//Timer Zurücksetzten.
		LTi_Zustand := 100;					//In den Error Zustand gehen.
		wState := FB_TSRCom.wState;			//Den ENUM Wert Error angeben.
	ELSE
		IF LTfn_Timer.Q THEN					//Wenn der Timer Abgelaufen ist.
			LTi_Zustand := 100;				//In den Error Zustand gehen.
			wState := 20;					//Den ENUM Wert Error angeben.
			LTfn_Timer.IN := 0;
		END_IF
	END_IF
LTfn_Timer(IN := 1, PT:= LCt_WaitTimeout);	//Setzte den Timer.
END_IF
LTfn_Timer();									//Timer Aufrufen.
END_ACTION

ACTION A6_Wait_for_TSR_Auswerten:
IF FB_TSRCom.stReceivedData = 'ready' THEN 		//Wenn der TSR reagiert.
	LTi_Zustand := 7;							//Gehe zum letzten Zustand.
	FB_TSRCom.xEXecute := 0;					//Setzte Com Communication zurück.
ELSE
	IF FB_TSRCom.stReceivedData = 'busy' THEN	//Wenn der TSR noch busy ist frage nochmal.
		FB_TSRCom.xEXecute := 0;				
		LTi_zustand := 4;
	ELSE
		IF FB_TSRCom.stReceivedData = '' THEN
			FB_TSRCom.xEXecute := 0;				
			LTi_zustand := 4;
		ELSE
			LTi_Zustand := 100;
			wState := 8;							//Gehe zum letzten Zustand.
		END_IF 
	END_IF
END_IF
END_ACTION

ACTION A7_End:
xBusy := 0;							//Alles zurücksetzten
xDone := 1;
IF xExecute = 0 THEN				//Warten bis der User Zurückgesetzt hat.
	xDone := 0;
	LTi_Zustand := 0;
	FB_TSRCom.xEXecute := 0;
END_IF
END_ACTION

ACTION B100_Error:
xBusy := 0;							//Alles zurücksetzten
xError := 1;
IF xExecute = 0 THEN				//Wartem bis der User das xExecute zurückgesetzt hat.
	xError := 0;
	LTi_Zustand := 0;
	wState := 0;					
	FB_TSRCom.xEXecute := 0;		//FB Com zurücksetzetn
END_IF
END_ACTION

END_FUNCTION_BLOCK

// POUs/FB Get TSR position/FB_Get_TSR_position
FUNCTION_BLOCK FB_Get_TSR_position
VAR_INPUT								//FB Eingänge
	xExecute				:BOOL;			//Startbedingung für den FB.
END_VAR

VAR_OUTPUT								//FB Ausgänge
	xBusy					:BOOL;			//Das Busy bit.
	xDone					:BOOL;			//Ist 1 wenn FB fertig ist.
	wState					:WORD;			//Der ENUM Wert für die ENUM Tabelle.
	xError					:BOOL;			//Ist 1 wenn es einen Error gab.
	iPosx					:INT;			//Die Position vom TSR.
	iPosy					:INT;			//Die Position vom TSR.
END_VAR

VAR										//Interne VAR
	LTi_Zustand				:INT;			//Der Zustand.
	LTi_PosMid				:INT;			//Diese Variable soll angeben bei welcher Position sich das : vom rückgabe wert befindet.
	LTi_Len					:INT;			//Gibt die String länge an für den Progress.
										//TIMER
	LTfn_Timer				:TON;			//Timer Init.
END_VAR

VAR CONSTANT							//Konstanten, Einstellung
	LCt_WaitTimeout		:TIME := T#2S;		//der Timout Timer.
END_VAR

CASE LTi_Zustand OF
	0:
		A0_Start();					//Prüfe Startbedingunen
	1:
		A1_Progress();				//Starte den Prozess. und sende den Befehl an das TSR.
	2:
		A2_Progress_Wait();			//Warte auf den FB Com.
	3:
		A3_Auswerten();				//Beende den FB und warte auf den User.
	4:
		A4_End();					//Das ende der Funktion.
	100:
		B100_Error();				//Die Error Aktion.
END_CASE

FB_TSRCom();						//Aufrufen.

ACTION A0_Start:
IF xExecute THEN			//Prüfe Startbedinung.
	xBusy := 1;				//Setze Busy.
	LTi_Zustand := 1;		//nächster Schritt
END_IF
END_ACTION

ACTION A1_Progress:
//TSR Com Aufrufen und Daten übergeben.
FB_TSRCom(						
	iCom		:= 1,
	xEXecute	:= 1, 
	stSendData	:= 	'getpos',);

//Auf zum nächsten schritt.
LTi_Zustand := 2;
END_ACTION

ACTION A2_Progress_Wait:
IF FB_TSRCom.xDone THEN						//Wenn der Port offen
	LTfn_Timer.IN := 0;						//Timer Zurücksetzten.
	LTi_Zustand := 3;						//Gehe in den Sende Schritt
ELSE
	IF FB_TSRCom.xError THEN				//Wenn es einen Error bei Com Port öffnen gab.
		LTfn_Timer.IN := 0;					//Timer Zurücksetzten.
		LTi_Zustand := 100;					//In den Error Zustand gehen.
		wState := FB_TSRCom.wState;			//Den ENUM Wert Error angeben.
	ELSE
		IF LTfn_Timer.Q THEN				//Wenn der Timer Abgelaufen ist.
			LTi_Zustand := 100;				//In den Error Zustand gehen.
			wState := 19;					//Den ENUM Wert Error angeben.
			LTfn_Timer.IN := 0;
		END_IF
	END_IF
LTfn_Timer(IN := 1, PT:= LCt_WaitTimeout);	//Setzte den Timer.
END_IF
LTfn_Timer();								//Timer Aufrufen.
END_ACTION

ACTION A3_Auswerten:
LTi_PosMid := FIND(FB_TSRCom.stReceivedData,':');	//Speichert die Pos wo sich das : befindet.
LTi_Len	:=	LEN(FB_TSRCom.stReceivedData);
iPosx := REAL_TO_INT(INT_TO_REAL((STRING_TO_INT(LEFT(STR:=FB_TSRCom.stReceivedData , SIZE:=LTi_PosMid))) - iStartPosx) / GTr_Faktor);
iPosy := REAL_TO_INT(INT_TO_REAL((STRING_TO_INT(RIGHT(STR:=FB_TSRCom.stReceivedData , SIZE:=LTi_Len - LTi_PosMid))) - iStartPosy) / GTr_Faktor);
LTi_Zustand := 4;
END_ACTION

ACTION A4_End:
xBusy := 0;							//Alles zurücksetzten
xDone := 1;
IF xExecute = 0 THEN				//Warten bis der User Zurückgesetzt hat.
	xDone := 0;
	LTi_Zustand := 0;
	FB_TSRCom.xEXecute := 0;
	iPosx := 0;
	iPosy := 0;
END_IF
END_ACTION

ACTION B100_Error:
xBusy := 0;							//Alles zurücksetzten
xError := 1;
IF xExecute = 0 THEN				//Wartem bis der User das xExecute zurückgesetzt hat.
	xError := 0;
	LTi_Zustand := 0;
	wState := 0;					
	FB_TSRCom.xEXecute := 0;		//FB Com zurücksetzetn
	iPosx := 0;
	iPosy := 0;
END_IF
END_ACTION

END_FUNCTION_BLOCK

// POUs/FB TSR Pen up down/TSR_Pen_up_down
FUNCTION_BLOCK TSR_Pen_up_down
VAR_INPUT								//Eingänge Var
	xExecute				:BOOL;			//Startbedingung für den FB.
	xPen					:BOOL;			//Wenn null = oben. und 1 = unten.
END_VAR

VAR_OUTPUT								//Ausgänge Var
	xBusy					:BOOL;			//Das Busy bit.
	xDone					:BOOL;			//Ist 1 wenn FB fertig ist.
	wState					:WORD;			//Der ENUM Wert für die ENUM Tabelle.
	xError					:BOOL;			//Ist 1 wenn es einen Error gab.
END_VAR

VAR										//Interne Var
	LTi_Zustand				:INT;			//Der Zustand.
	LTst_String				:STRING;		//Ein Zwischenspeicher.
										//TIMER
	LTfn_Timer				:TON;			//Timer Init
END_VAR

VAR CONSTANT							//Konstanten, Einstellungen
	LCt_WaitTimeout		:TIME := T#2S;		//der Timout Timer.
END_VAR

CASE LTi_Zustand OF
	0:
		A0_Start();					//Prüfe die Startbedingungen 
	1:
		A1_Progress();				//Starte den Prozess.
	2:
		A2_Progress_Wait();			//Warte auf den FB TSR Com
	3:
		A3_Auswerten();				//Werte das Egebniss aus.
	4:
		A4_End();					//Warte auf Execute
	100:
		B100_Error();				//Nur wenn ein Error gab.
END_CASE

FB_TSRCom();

ACTION A0_Start:
IF xExecute THEN			//Prüfe Startbedinung.
	xBusy := 1;				//Setze Busy.
	LTi_Zustand := 1;	//Gehe direkt zum Schritt wo der Com Port geöffnet wird.
END_IF
END_ACTION

ACTION A1_Progress:
IF xPen THEN
	LTst_String := 'touchdown';
ELSE
	LTst_String := 'touchup';
END_IF


FB_TSRCom(						//TSR Com Aufrufen und Daten übergeben.
	xEXecute	:=	1 ,  
	stSendData	:= 	LTst_String,  );
LTi_Zustand := 2;				//In den nächsten Zustand Wechseln.
END_ACTION

ACTION A2_Progress_Wait:
IF FB_TSRCom.xDone THEN											//Wenn der Port offen
	LTfn_Timer.IN := 0;					//Timer Zurücksetzten.
	LTi_Zustand := 3;					//Gehe in den Sende Schritt
ELSE
	IF FB_TSRCom.xError THEN				//Wenn es einen Error bei Com Port öffnen gab.
		LTfn_Timer.IN := 0;					//Timer Zurücksetzten.
		LTi_Zustand := 100;					//In den Error Zustand gehen.
		wState := FB_TSRCom.wState;			//Den ENUM Wert Error angeben.
	ELSE
		IF LTfn_Timer.Q THEN						//Wenn der Timer Abgelaufen ist.
			LTi_Zustand := 100;					//In den Error Zustand gehen.
			wState := 22;						//Den ENUM Wert Error angeben.
			LTfn_Timer.IN := 0;
		END_IF
	END_IF
LTfn_Timer(IN := 1, PT:= LCt_WaitTimeout);
END_IF

LTfn_Timer();								//Rufe Timer auf
END_ACTION

ACTION A3_Auswerten:
IF FB_TSRCom.stReceivedData = 'ok' THEN		//Wenn der TSR reagiert.
	LTi_Zustand := 4;						//Gehe zum letzten Zustand.
ELSE											
	LTi_Zustand := 100;	
	wState := 8;								
END_IF
END_ACTION

ACTION A4_End:
xBusy := 0;							//Alles zurücksetzten
xDone := 1;
IF xExecute = 0 THEN				//Warten bis der User Zurückgesetzt hat.
	xDone := 0;
	LTi_Zustand := 0;
	FB_TSRCom.xEXecute := 0;
END_IF
END_ACTION

ACTION B100_Error:
xBusy := 0;							//Alles zurücksetzten
xError := 1;
IF xExecute = 0 THEN				//Wartem bis der User das xExecute zurückgesetzt hat.
	xError := 0;
	LTi_Zustand := 0;
	wState := 0;
	FB_TSRCom.xEXecute := 0;
END_IF
END_ACTION

END_FUNCTION_BLOCK

// POUs/FB Click/FB_Click
FUNCTION_BLOCK FB_Click
VAR_INPUT
	xExecute		:BOOL;		//Startet den FB
	iKlicktox		:INT;		//Die x Koordinate für den Klick
	iKlicktoy		:INT;		//Die y Koordinate für den Klick
END_VAR

VAR_OUTPUT
	xBusy			:BOOL;					//Das busy bool
	xDone			:BOOL;					//Wenn der FB fertig ist
	wState			:WORD;					//Gibt den status im error fall an
	xError			:BOOL;					//Das Error Flag.
END_VAR

VAR
	LTfn_Timer		:TON;					//Timer Init.
	LTfb_Goto		:FB_Go_to_TSR_xy;		//Die GOTO Funktion aufrufen
	LTi_Zustand		:INT;					//Gibt den Zustand an den man benötigt.
	LCt_WaitTimeout	:TIME := T#4S;			//Die Timeout zeit.
	LTfb_Pen		:TSR_Pen_up_down;
END_VAR

CASE LTi_Zustand OF
	0:
		A0_Start();
	1:
		A1_Progress();
	2:
		A2_Progress_Wait();
	3:
		A3_PenDown();
	4:
		A4_PenDown_Wait();
	5:
		A5_PenUp();
	6:
		A6_PenUp_Wait();
	7:
		A7_End();
	100:
		B100_Error();
END_CASE
LTfb_Pen();
LTfb_Goto();
LTfn_Timer();

ACTION A0_Start:
IF xExecute THEN			//Prüfe Startbedinung.
	xBusy := 1;				//Setze Busy.
	LTi_Zustand := 1;		//nächster Schritt
END_IF

FB_TSRCom();				//Den Com aufrufen.
END_ACTION

ACTION A1_Progress:
LTfb_Goto
(
	xExecute := 1, 
	iGotox := iKlicktox , 
	iGotoy := iKlicktoy , 
);

LTi_Zustand := 2;
END_ACTION

ACTION A2_Progress_Wait:
IF LTfb_Goto.xDone THEN											//Wenn der Port offen
	LTfn_Timer.IN := 0;						//Timer Zurücksetzten.
	LTi_Zustand := 3;						//Gehe in den Sende Schritt
ELSE
	IF LTfb_Goto.xError THEN				//Wenn es einen Error bei Com Port öffnen gab.
		LTfn_Timer.IN := 0;					//Timer Zurücksetzten.
		LTi_Zustand := 100;					//In den Error Zustand gehen.
		wState := LTfb_Goto.wState;			//Den ENUM Wert Error angeben.
	ELSE
		IF LTfn_Timer.Q THEN				//Wenn der Timer Abgelaufen ist.
			LTi_Zustand := 100;				//In den Error Zustand gehen.
			wState := 14;					//Timeout beim Click Goto
			LTfn_Timer.IN := 0;
		END_IF
	END_IF
LTfn_Timer(IN := 1, PT:= LCt_WaitTimeout);	//Setzte den Timer.
END_IF
LTfn_Timer();								//Timer Aufrufen.
END_ACTION

ACTION A3_PenDown:
LTfb_Pen
(
	xExecute := 1, 
	xPen := 1, 
);

LTi_Zustand := 4;
END_ACTION

ACTION A4_PenDown_Wait:
IF LTfb_Pen.xDone THEN						//Wenn der Port offen
	LTfn_Timer.IN := 0;						//Timer Zurücksetzten.
	LTi_Zustand := 5;						//Gehe in den Sende Schritt
	LTfb_Pen.xExecute := 0;					//Den FB zurücksetzten
	LTfb_Pen();								//Denn FB aufrufen um zurückzusetzten.
ELSE
	IF LTfb_Pen.xError THEN					//Wenn es einen Error bei Com Port öffnen gab.
		LTfn_Timer.IN := 0;					//Timer Zurücksetzten.
		LTi_Zustand := 100;					//In den Error Zustand gehen.
		wState := LTfb_Pen.wState;			//Den ENUM Wert Error angeben.
	ELSE
		IF LTfn_Timer.Q THEN				//Wenn der Timer Abgelaufen ist.
			LTi_Zustand := 100;				//In den Error Zustand gehen.
			wState := 15;					//Den ENUM Wert Error angeben.
			LTfn_Timer.IN := 0;
		END_IF
	END_IF
LTfn_Timer(IN := 1, PT:= LCt_WaitTimeout);	//Setzte den Timer.
END_IF
LTfn_Timer();								//Timer Aufrufen.
END_ACTION

ACTION A5_PenUp:
LTfb_Pen
(
	xExecute := 1, 
	xPen := 0, 
);

LTi_Zustand := 6;
END_ACTION

ACTION A6_PenUp_Wait:
IF LTfb_Pen.xDone THEN						//Wenn der Port offen
	LTfn_Timer.IN := 0;						//Timer Zurücksetzten.
	LTi_Zustand := 7;						//Gehe in den Sende Schritt
ELSE
	IF LTfb_Pen.xError THEN					//Wenn es einen Error bei Com Port öffnen gab.
		LTfn_Timer.IN := 0;					//Timer Zurücksetzten.
		LTi_Zustand := 100;					//In den Error Zustand gehen.
		wState := LTfb_Pen.wState;			//Den ENUM Wert Error angeben.
	ELSE
		IF LTfn_Timer.Q THEN				//Wenn der Timer Abgelaufen ist.
			LTi_Zustand := 100;				//In den Error Zustand gehen.
			wState := 15;					//Den ENUM Wert Error angeben.
			LTfn_Timer.IN := 0;
		END_IF
	END_IF
LTfn_Timer(IN := 1, PT:= LCt_WaitTimeout);	//Setzte den Timer.
END_IF
LTfn_Timer();								//Timer Aufrufen.
END_ACTION

ACTION A7_End:
xBusy := 0;							//Alles zurücksetzten
xDone := 1;
IF xExecute = 0 THEN				//Warten bis der User Zurückgesetzt hat.
	xDone := 0;
	LTi_Zustand := 0;
	lTfb_Pen.xEXecute := 0;
	lTfb_Goto.xEXecute := 0;
END_IF
END_ACTION

ACTION B100_Error:
xBusy := 0;							//Alles zurücksetzten
xError := 1;
IF xExecute = 0 THEN				//Wartem bis der User das xExecute zurückgesetzt hat.
	xError := 0;
	LTi_Zustand := 0;
	wState := 0;					
	LTfb_Pen.xEXecute := 0;		//FB Com zurücksetzetn.
	LTfb_Goto.xEXecute := 0;	//FB GOTO zurüksetzen.
END_IF
END_ACTION

END_FUNCTION_BLOCK

// POUs/FB Double Click/FB_Double_Click
FUNCTION_BLOCK FB_Double_Click
VAR_INPUT
	xExecute		:BOOL;		//Startet den FB
	iKlicktox		:INT;		//Die x Koordinate für den Klick
	iKlicktoy		:INT;		//Die y Koordinate für den Klick
END_VAR

VAR_OUTPUT
	xBusy			:BOOL;					//Das busy bool
	xDone			:BOOL;					//Wenn der FB fertig ist
	wState			:WORD;					//Gibt den status im error fall an
	xError			:BOOL;					//Das Error Flag.
END_VAR

VAR
	LTfn_Timer		:TON;					//Timer Init.
	LTfb_Goto		:FB_Go_to_TSR_xy;		//Die GOTO Funktion aufrufen
	LTi_Zustand		:INT;					//Gibt den Zustand an den man benötigt.
	LCt_WaitTimeout	:TIME := T#4S;			//Die Timeout zeit.
	LTfb_Pen		:TSR_Pen_up_down;
	LTx_FirstTime	:BOOL;					//First TIme Bool damit man 2 mal Klickt.
END_VAR

CASE LTi_Zustand OF
	0:
		A0_Start();
	1:
		A1_Progress();
	2:
		A2_Progress_Wait();
	3:
		A3_PenDown();
	4:
		A4_PenDown_Wait();
	5:
		A5_PenUp();
	6:
		A6_PenUp_Wait();
	7:
		A7_End();
	100:
		B100_Error();
END_CASE
LTfb_Pen();
LTfb_Goto();

ACTION A0_Start:
IF xExecute THEN			//Prüfe Startbedinung.
	xBusy := 1;				//Setze Busy.
	LTi_Zustand := 1;		//nächster Schritt
END_IF
END_ACTION

ACTION A1_Progress:
LTfb_Goto
(
	xExecute := 1, 
	iGotox := iKlicktox , 
	iGotoy := iKlicktoy , 
);

LTi_Zustand := 2;
END_ACTION

ACTION A2_Progress_Wait:
IF LTfb_Goto.xDone THEN											//Wenn der Port offen
	LTfn_Timer.IN := 0;						//Timer Zurücksetzten.
	LTi_Zustand := 3;						//Gehe in den Sende Schritt
ELSE
	IF LTfb_Goto.xError THEN				//Wenn es einen Error bei Com Port öffnen gab.
		LTfn_Timer.IN := 0;					//Timer Zurücksetzten.
		LTi_Zustand := 100;					//In den Error Zustand gehen.
		wState := LTfb_Goto.wState;			//Den ENUM Wert Error angeben.
	ELSE
		IF LTfn_Timer.Q THEN				//Wenn der Timer Abgelaufen ist.
			LTi_Zustand := 100;				//In den Error Zustand gehen.
			wState := 17;					//Den ENUM Wert Error angeben.
			LTfn_Timer.IN := 0;
		END_IF
	END_IF
LTfn_Timer(IN := 1, PT:= LCt_WaitTimeout);	//Setzte den Timer.
END_IF
LTfn_Timer();								//Timer Aufrufen.
END_ACTION

ACTION A3_PenDown:
LTfb_Pen
(
	xExecute := 1, 
	xPen := 1, 
);

LTi_Zustand := 4;
END_ACTION

ACTION A4_PenDown_Wait:
IF LTfb_Pen.xDone THEN						//Wenn der Port offen
	LTfn_Timer.IN := 0;						//Timer Zurücksetzten.
	LTi_Zustand := 5;						//Gehe in den Sende Schritt
	LTfb_Pen.xExecute := 0;					//Den FB zurücksetzten
	LTfb_Pen();								//Denn FB aufrufen um zurückzusetzten.
ELSE
	IF LTfb_Pen.xError THEN					//Wenn es einen Error bei Com Port öffnen gab.
		LTfn_Timer.IN := 0;					//Timer Zurücksetzten.
		LTi_Zustand := 100;					//In den Error Zustand gehen.
		wState := LTfb_Pen.wState;			//Den ENUM Wert Error angeben.
	ELSE
		IF LTfn_Timer.Q THEN				//Wenn der Timer Abgelaufen ist.
			LTi_Zustand := 100;				//In den Error Zustand gehen.
			wState := 18;					//Den ENUM Wert Error angeben.
			LTfn_Timer.IN := 0;
		END_IF
	END_IF
LTfn_Timer(IN := 1, PT:= LCt_WaitTimeout);	//Setzte den Timer.
END_IF
LTfn_Timer();								//Timer Aufrufen.
END_ACTION

ACTION A5_PenUp:
LTfb_Pen
(
	xExecute := 1, 
	xPen := 0, 
);

LTi_Zustand := 6;
END_ACTION

ACTION A6_PenUp_Wait:
IF LTfb_Pen.xDone THEN						//Wenn der Port offen
	LTfn_Timer.IN := 0;						//Timer Zurücksetzten.
	IF LTx_FirstTime = 0 THEN
		LTi_Zustand := 3;
		LTfb_Pen.xExecute := 0;
		LTx_FirstTime := 1;
	ELSE
		LTi_Zustand := 7;					//Gehe in den Sende Schritt	
	END_IF
ELSE
	IF LTfb_Pen.xError THEN					//Wenn es einen Error bei Com Port öffnen gab.
		LTfn_Timer.IN := 0;					//Timer Zurücksetzten.
		LTi_Zustand := 100;					//In den Error Zustand gehen.
		wState := LTfb_Pen.wState;			//Den ENUM Wert Error angeben.
	ELSE
		IF LTfn_Timer.Q THEN				//Wenn der Timer Abgelaufen ist.
			LTi_Zustand := 100;				//In den Error Zustand gehen.
			wState := 18;					//Den ENUM Wert Error angeben.
			LTfn_Timer.IN := 0;
		END_IF
	END_IF
LTfn_Timer(IN := 1, PT:= LCt_WaitTimeout);	//Setzte den Timer.
END_IF
LTfn_Timer();								//Timer Aufrufen.
END_ACTION

ACTION A7_End:
xBusy := 0;							//Alles zurücksetzten
xDone := 1;
IF xExecute = 0 THEN				//Warten bis der User Zurückgesetzt hat.
	xDone := 0;
	LTi_Zustand := 0;
	lTfb_Pen.xEXecute := 0;
	lTfb_Goto.xEXecute := 0;
	LTx_FirstTime := 0;
END_IF
END_ACTION

ACTION B100_Error:
xBusy := 0;							//Alles zurücksetzten
xError := 1;
IF xExecute = 0 THEN				//Wartem bis der User das xExecute zurückgesetzt hat.
	xError := 0;
	LTi_Zustand := 0;
	wState := 0;					
	LTfb_Pen.xEXecute := 0;		//FB Com zurücksetzetn.
	LTfb_Goto.xEXecute := 0;	//FB GOTO zurüksetzen.
	LTx_FirstTime := 0;
END_IF
END_ACTION

END_FUNCTION_BLOCK
